(* PLC project Unnamed, Unknown Unnamed 1 *)
(* stored: creationDateTime 2022-07-16T10:46:25, modificationDateTime 2022-07-16T22:47:46 *)

PROGRAM program0
  VAR
    LocalVar0 AT %IL0.0 : LREAL;
    LocalVar1 AT %QL0.0 : LREAL;
  END_VAR
  VAR
    python_poll0 : python_poll;
  END_VAR

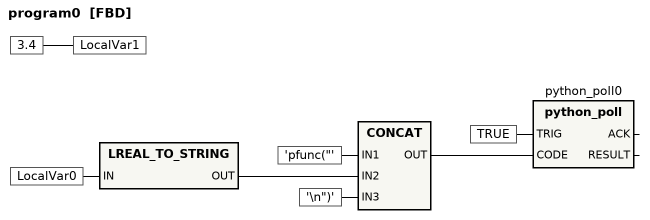
(* FBD diagram, written out as Structured Text *)
LocalVar1 := 3.4;
python_poll0(TRIG := TRUE, CODE := CONCAT('pfunc("', LREAL_TO_STRING(LocalVar0), '\n")'));
END_PROGRAM

CONFIGURATION config
  RESOURCE resource1 ON PLC
    TASK task0(INTERVAL := T#100ms, PRIORITY := 0);
    PROGRAM instance0 WITH task0 : program0;
  END_RESOURCE
END_CONFIGURATION
